// Extracts the underlying object pointer from an interface pointer.
// [note] The interface must inherit from __SYSTEM.IQueryInterface, otherwise the check is not valid.
FUNCTION F_ExtractPointerFromInterface : POINTER TO BYTE // Returns pointer to the concrete object or 0 if invalid.
VAR_INPUT
	// Address of the interface (e.g. ADR(ipInterface)).
	pInterface : POINTER TO BYTE;
END_VAR
VAR
	pTmp : POINTER TO POINTER TO BYTE := pInterface;
END_VAR

RETURN( NOT(F_IsReadablePointer(pInterface) AND F_IsPointerToInterface(pInterface)) );

F_ExtractPointerFromInterface := pTmp^;

END_FUNCTION

(* stored: Version 1.1.0.1
   POU F_ExtractPointerFromInterface: Id {ca5a1699-7c93-0173-3269-b173b8a5ed2d}, SpecialFunc None *)
